// TIA Portal V17 export
// export: Created 2025-06-26T07:49:56.8755819Z, ExportSetting WithDefaults, DisplayName Totally Integrated Automation Portal, DisplayVersion V17 Update 8, DisplayName TIA Portal Openness, DisplayVersion V17 Update 8, DisplayName TIA Portal Version Control Interface, DisplayVersion V17, DisplayName STEP 7 Professional, DisplayVersion V17 Update 8, DisplayName STEP 7 Safety, DisplayVersion V17 Update 6, DisplayName WinCC Advanced, DisplayVersion V17 Update 8
TYPE "stOilRecovery"
// stored: IsFailsafeCompliant false
   STRUCT
      bEnable : Bool;   // Run signal. 1 = Run, 0 = do not run
      nRunRatio : UInt;   // Run once every X times Run signal is active
      fFixedOutput : Real;   // [%] Valve setting when active
      fOut : Real;   // [%] Actual output
      Controller : "stOneShotRegulator";
   END_STRUCT;
END_TYPE
